// TIA Portal V18 export
FUNCTION "TEMPLATE--v1.1--05_Output Feedback" : Void   // FC6, F_FBD
TITLE = Manage Safety Outputs
{ S7_Optimized_Access := 'TRUE' }
// v1.0 First Emission
// v1.1 Added 03_FDBACK_RAW reference
   VAR_TEMP
      DU_EX : Bool;
      ISPC_EX : Bool;
      ZONE_EX : Bool;
   END_VAR
BEGIN

REGION Network 1: !!NetworkComment$$ 1c -1i -1q
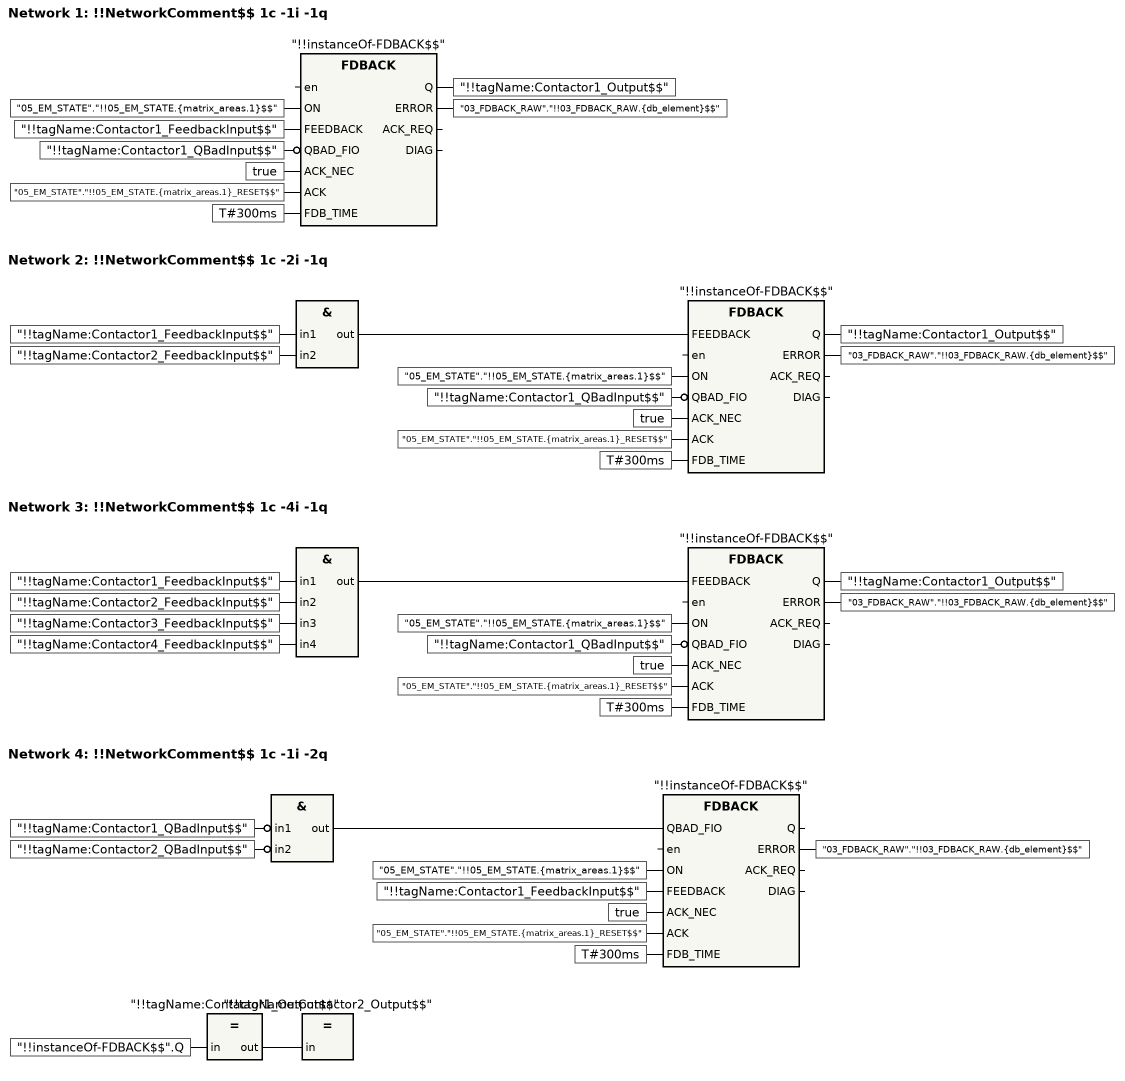
   "!!instanceOf-FDBACK$$"(ON := "05_EM_STATE"."!!05_EM_STATE.{matrix_areas.1}$$",   // FDBACK
                           FEEDBACK := "!!tagName:Contactor1_FeedbackInput$$",
                           QBAD_FIO := NOT "!!tagName:Contactor1_QBadInput$$",
                           ACK_NEC := true,
                           ACK := "05_EM_STATE"."!!05_EM_STATE.{matrix_areas.1}_RESET$$",
                           FDB_TIME := T#300ms,
                           Q => "!!tagName:Contactor1_Output$$",
                           ERROR => "03_FDBACK_RAW"."!!03_FDBACK_RAW.{db_element}$$");
END_REGION

REGION Network 2: !!NetworkComment$$ 1c -2i -1q
   "!!instanceOf-FDBACK$$"(FEEDBACK := "!!tagName:Contactor1_FeedbackInput$$" AND "!!tagName:Contactor2_FeedbackInput$$",   // FDBACK
                           ON := "05_EM_STATE"."!!05_EM_STATE.{matrix_areas.1}$$",
                           QBAD_FIO := NOT "!!tagName:Contactor1_QBadInput$$",
                           ACK_NEC := true,
                           ACK := "05_EM_STATE"."!!05_EM_STATE.{matrix_areas.1}_RESET$$",
                           FDB_TIME := T#300ms,
                           Q => "!!tagName:Contactor1_Output$$",
                           ERROR => "03_FDBACK_RAW"."!!03_FDBACK_RAW.{db_element}$$");
END_REGION

REGION Network 3: !!NetworkComment$$ 1c -4i -1q
   "!!instanceOf-FDBACK$$"(FEEDBACK := "!!tagName:Contactor1_FeedbackInput$$" AND "!!tagName:Contactor2_FeedbackInput$$" AND "!!tagName:Contactor3_FeedbackInput$$" AND "!!tagName:Contactor4_FeedbackInput$$",   // FDBACK
                           ON := "05_EM_STATE"."!!05_EM_STATE.{matrix_areas.1}$$",
                           QBAD_FIO := NOT "!!tagName:Contactor1_QBadInput$$",
                           ACK_NEC := true,
                           ACK := "05_EM_STATE"."!!05_EM_STATE.{matrix_areas.1}_RESET$$",
                           FDB_TIME := T#300ms,
                           Q => "!!tagName:Contactor1_Output$$",
                           ERROR => "03_FDBACK_RAW"."!!03_FDBACK_RAW.{db_element}$$");
END_REGION

REGION Network 4: !!NetworkComment$$ 1c -1i -2q
   "!!instanceOf-FDBACK$$"(QBAD_FIO := NOT "!!tagName:Contactor1_QBadInput$$" AND NOT "!!tagName:Contactor2_QBadInput$$",   // FDBACK
                           ON := "05_EM_STATE"."!!05_EM_STATE.{matrix_areas.1}$$",
                           FEEDBACK := "!!tagName:Contactor1_FeedbackInput$$",
                           ACK_NEC := true,
                           ACK := "05_EM_STATE"."!!05_EM_STATE.{matrix_areas.1}_RESET$$",
                           FDB_TIME := T#300ms,
                           ERROR => "03_FDBACK_RAW"."!!03_FDBACK_RAW.{db_element}$$");
   "!!tagName:Contactor1_Output$$" := "!!instanceOf-FDBACK$$".Q;
   "!!tagName:Contactor2_Output$$" := "!!instanceOf-FDBACK$$".Q;
END_REGION

REGION Network 5: !!NetworkComment$$ 1c -2i -2q
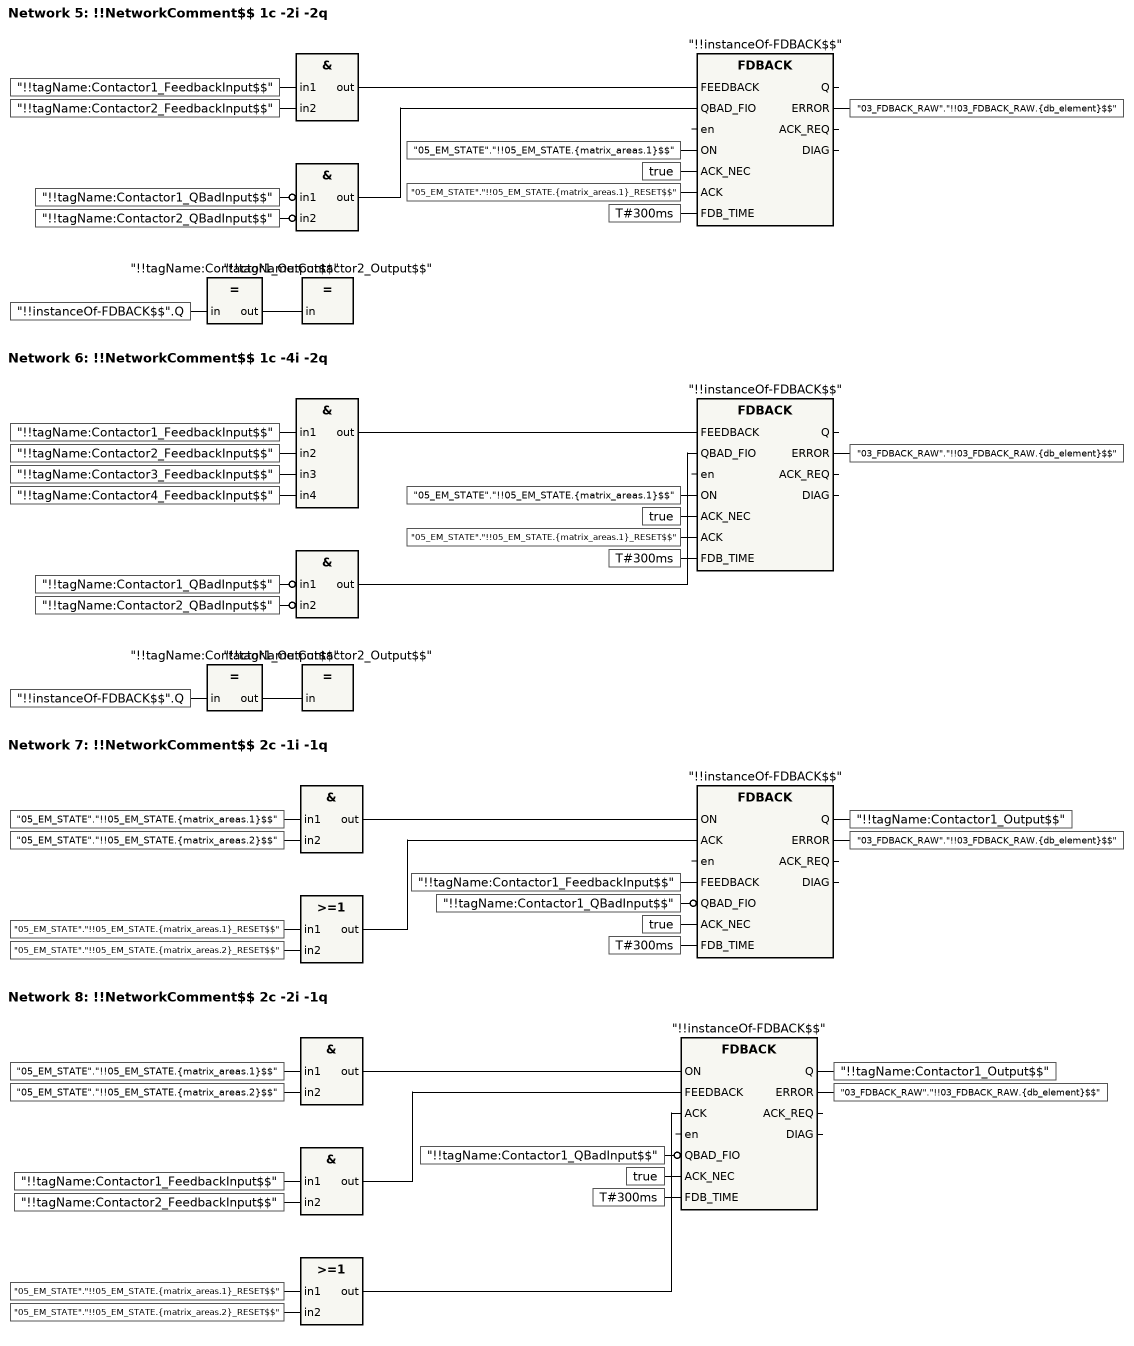
   "!!instanceOf-FDBACK$$"(FEEDBACK := "!!tagName:Contactor1_FeedbackInput$$" AND "!!tagName:Contactor2_FeedbackInput$$",   // FDBACK
                           QBAD_FIO := NOT "!!tagName:Contactor1_QBadInput$$" AND NOT "!!tagName:Contactor2_QBadInput$$",
                           ON := "05_EM_STATE"."!!05_EM_STATE.{matrix_areas.1}$$",
                           ACK_NEC := true,
                           ACK := "05_EM_STATE"."!!05_EM_STATE.{matrix_areas.1}_RESET$$",
                           FDB_TIME := T#300ms,
                           ERROR => "03_FDBACK_RAW"."!!03_FDBACK_RAW.{db_element}$$");
   "!!tagName:Contactor1_Output$$" := "!!instanceOf-FDBACK$$".Q;
   "!!tagName:Contactor2_Output$$" := "!!instanceOf-FDBACK$$".Q;
END_REGION

REGION Network 6: !!NetworkComment$$ 1c -4i -2q
   "!!instanceOf-FDBACK$$"(FEEDBACK := "!!tagName:Contactor1_FeedbackInput$$" AND "!!tagName:Contactor2_FeedbackInput$$" AND "!!tagName:Contactor3_FeedbackInput$$" AND "!!tagName:Contactor4_FeedbackInput$$",   // FDBACK
                           QBAD_FIO := NOT "!!tagName:Contactor1_QBadInput$$" AND NOT "!!tagName:Contactor2_QBadInput$$",
                           ON := "05_EM_STATE"."!!05_EM_STATE.{matrix_areas.1}$$",
                           ACK_NEC := true,
                           ACK := "05_EM_STATE"."!!05_EM_STATE.{matrix_areas.1}_RESET$$",
                           FDB_TIME := T#300ms,
                           ERROR => "03_FDBACK_RAW"."!!03_FDBACK_RAW.{db_element}$$");
   "!!tagName:Contactor1_Output$$" := "!!instanceOf-FDBACK$$".Q;
   "!!tagName:Contactor2_Output$$" := "!!instanceOf-FDBACK$$".Q;
END_REGION

REGION Network 7: !!NetworkComment$$ 2c -1i -1q
   "!!instanceOf-FDBACK$$"(ON := "05_EM_STATE"."!!05_EM_STATE.{matrix_areas.1}$$" AND "05_EM_STATE"."!!05_EM_STATE.{matrix_areas.2}$$",   // FDBACK
                           ACK := "05_EM_STATE"."!!05_EM_STATE.{matrix_areas.1}_RESET$$" OR "05_EM_STATE"."!!05_EM_STATE.{matrix_areas.2}_RESET$$",
                           FEEDBACK := "!!tagName:Contactor1_FeedbackInput$$",
                           QBAD_FIO := NOT "!!tagName:Contactor1_QBadInput$$",
                           ACK_NEC := true,
                           FDB_TIME := T#300ms,
                           Q => "!!tagName:Contactor1_Output$$",
                           ERROR => "03_FDBACK_RAW"."!!03_FDBACK_RAW.{db_element}$$");
END_REGION

REGION Network 8: !!NetworkComment$$ 2c -2i -1q
   "!!instanceOf-FDBACK$$"(ON := "05_EM_STATE"."!!05_EM_STATE.{matrix_areas.1}$$" AND "05_EM_STATE"."!!05_EM_STATE.{matrix_areas.2}$$",   // FDBACK
                           FEEDBACK := "!!tagName:Contactor1_FeedbackInput$$" AND "!!tagName:Contactor2_FeedbackInput$$",
                           ACK := "05_EM_STATE"."!!05_EM_STATE.{matrix_areas.1}_RESET$$" OR "05_EM_STATE"."!!05_EM_STATE.{matrix_areas.2}_RESET$$",
                           QBAD_FIO := NOT "!!tagName:Contactor1_QBadInput$$",
                           ACK_NEC := true,
                           FDB_TIME := T#300ms,
                           Q => "!!tagName:Contactor1_Output$$",
                           ERROR => "03_FDBACK_RAW"."!!03_FDBACK_RAW.{db_element}$$");
END_REGION

REGION Network 9: !!NetworkComment$$ 1c -4i -1q
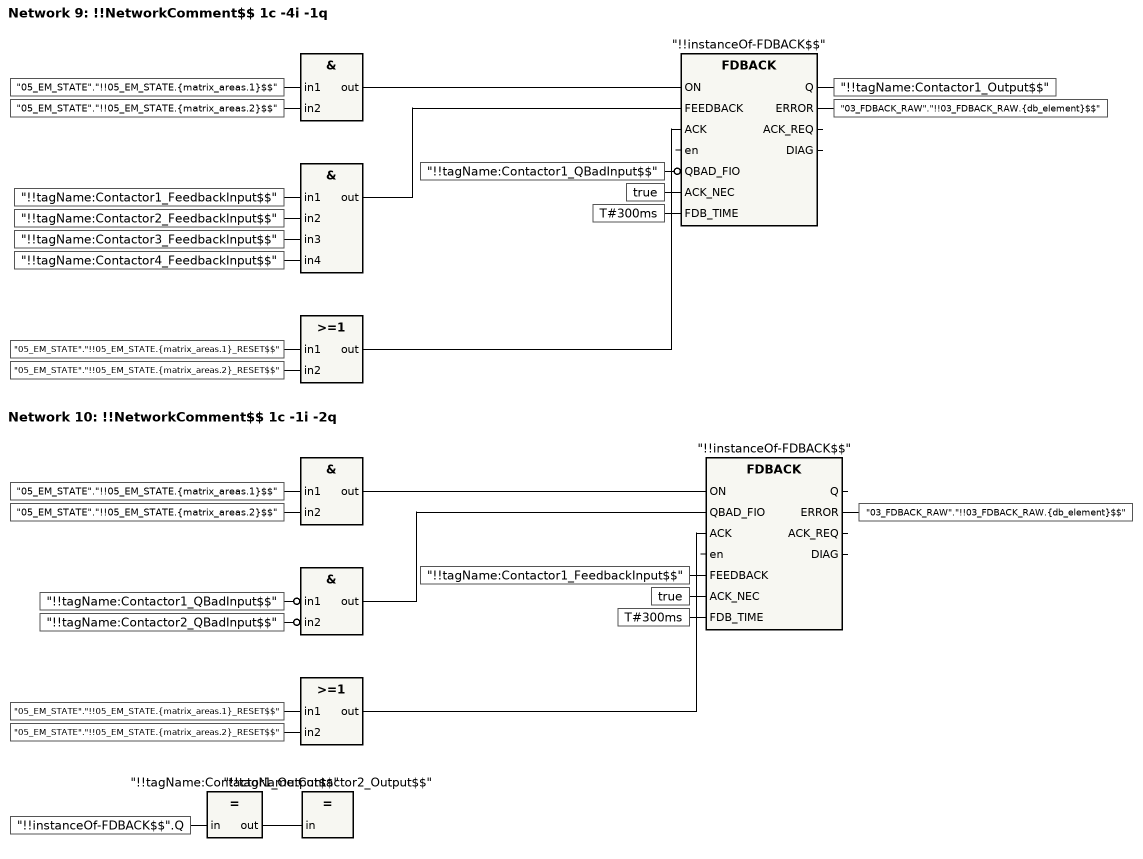
   "!!instanceOf-FDBACK$$"(ON := "05_EM_STATE"."!!05_EM_STATE.{matrix_areas.1}$$" AND "05_EM_STATE"."!!05_EM_STATE.{matrix_areas.2}$$",   // FDBACK
                           FEEDBACK := "!!tagName:Contactor1_FeedbackInput$$" AND "!!tagName:Contactor2_FeedbackInput$$" AND "!!tagName:Contactor3_FeedbackInput$$" AND "!!tagName:Contactor4_FeedbackInput$$",
                           ACK := "05_EM_STATE"."!!05_EM_STATE.{matrix_areas.1}_RESET$$" OR "05_EM_STATE"."!!05_EM_STATE.{matrix_areas.2}_RESET$$",
                           QBAD_FIO := NOT "!!tagName:Contactor1_QBadInput$$",
                           ACK_NEC := true,
                           FDB_TIME := T#300ms,
                           Q => "!!tagName:Contactor1_Output$$",
                           ERROR => "03_FDBACK_RAW"."!!03_FDBACK_RAW.{db_element}$$");
END_REGION

REGION Network 10: !!NetworkComment$$ 1c -1i -2q
   "!!instanceOf-FDBACK$$"(ON := "05_EM_STATE"."!!05_EM_STATE.{matrix_areas.1}$$" AND "05_EM_STATE"."!!05_EM_STATE.{matrix_areas.2}$$",   // FDBACK
                           QBAD_FIO := NOT "!!tagName:Contactor1_QBadInput$$" AND NOT "!!tagName:Contactor2_QBadInput$$",
                           ACK := "05_EM_STATE"."!!05_EM_STATE.{matrix_areas.1}_RESET$$" OR "05_EM_STATE"."!!05_EM_STATE.{matrix_areas.2}_RESET$$",
                           FEEDBACK := "!!tagName:Contactor1_FeedbackInput$$",
                           ACK_NEC := true,
                           FDB_TIME := T#300ms,
                           ERROR => "03_FDBACK_RAW"."!!03_FDBACK_RAW.{db_element}$$");
   "!!tagName:Contactor1_Output$$" := "!!instanceOf-FDBACK$$".Q;
   "!!tagName:Contactor2_Output$$" := "!!instanceOf-FDBACK$$".Q;
END_REGION

REGION Network 11: !!NetworkComment$$ 1c -2i -2q
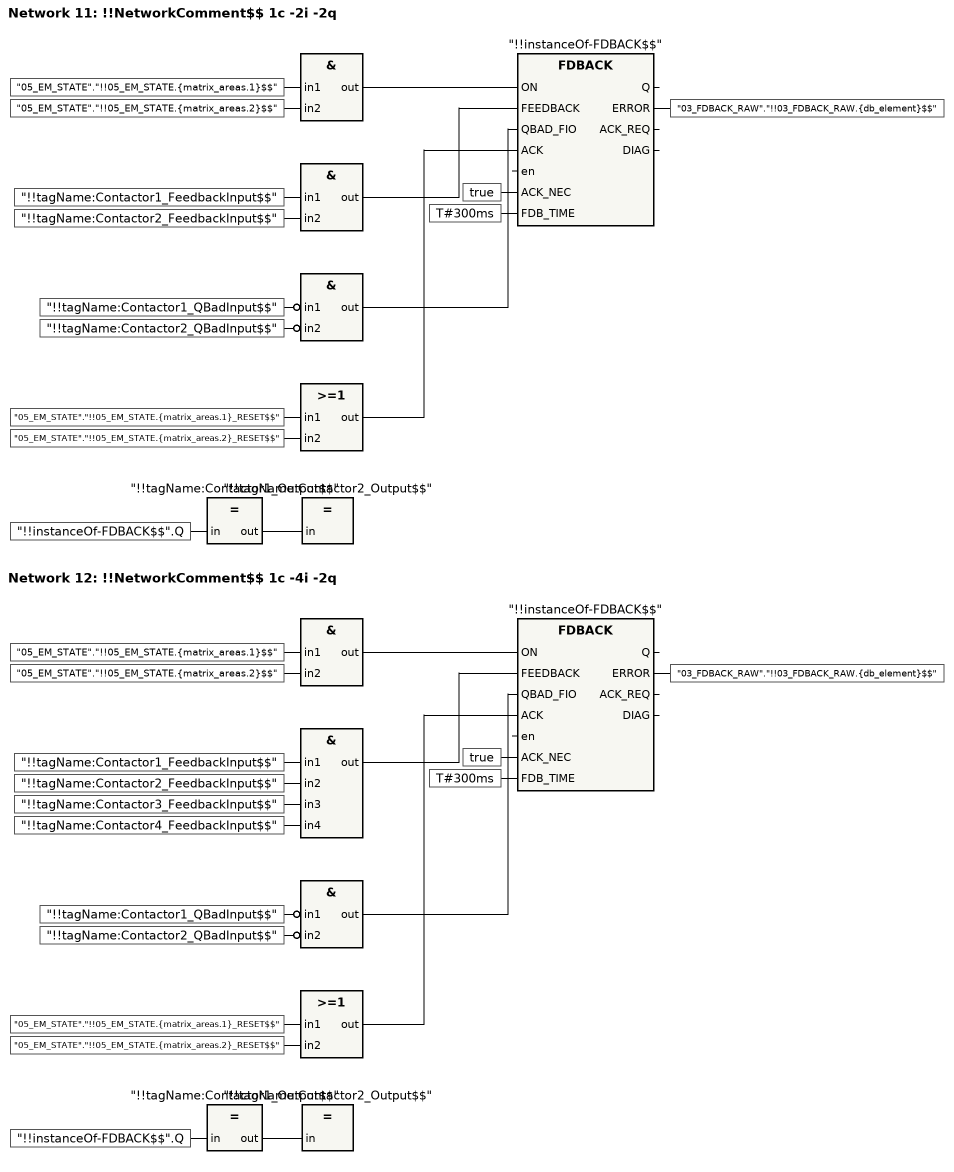
   "!!instanceOf-FDBACK$$"(ON := "05_EM_STATE"."!!05_EM_STATE.{matrix_areas.1}$$" AND "05_EM_STATE"."!!05_EM_STATE.{matrix_areas.2}$$",   // FDBACK
                           FEEDBACK := "!!tagName:Contactor1_FeedbackInput$$" AND "!!tagName:Contactor2_FeedbackInput$$",
                           QBAD_FIO := NOT "!!tagName:Contactor1_QBadInput$$" AND NOT "!!tagName:Contactor2_QBadInput$$",
                           ACK := "05_EM_STATE"."!!05_EM_STATE.{matrix_areas.1}_RESET$$" OR "05_EM_STATE"."!!05_EM_STATE.{matrix_areas.2}_RESET$$",
                           ACK_NEC := true,
                           FDB_TIME := T#300ms,
                           ERROR => "03_FDBACK_RAW"."!!03_FDBACK_RAW.{db_element}$$");
   "!!tagName:Contactor1_Output$$" := "!!instanceOf-FDBACK$$".Q;
   "!!tagName:Contactor2_Output$$" := "!!instanceOf-FDBACK$$".Q;
END_REGION

REGION Network 12: !!NetworkComment$$ 1c -4i -2q
   "!!instanceOf-FDBACK$$"(ON := "05_EM_STATE"."!!05_EM_STATE.{matrix_areas.1}$$" AND "05_EM_STATE"."!!05_EM_STATE.{matrix_areas.2}$$",   // FDBACK
                           FEEDBACK := "!!tagName:Contactor1_FeedbackInput$$" AND "!!tagName:Contactor2_FeedbackInput$$" AND "!!tagName:Contactor3_FeedbackInput$$" AND "!!tagName:Contactor4_FeedbackInput$$",
                           QBAD_FIO := NOT "!!tagName:Contactor1_QBadInput$$" AND NOT "!!tagName:Contactor2_QBadInput$$",
                           ACK := "05_EM_STATE"."!!05_EM_STATE.{matrix_areas.1}_RESET$$" OR "05_EM_STATE"."!!05_EM_STATE.{matrix_areas.2}_RESET$$",
                           ACK_NEC := true,
                           FDB_TIME := T#300ms,
                           ERROR => "03_FDBACK_RAW"."!!03_FDBACK_RAW.{db_element}$$");
   "!!tagName:Contactor1_Output$$" := "!!instanceOf-FDBACK$$".Q;
   "!!tagName:Contactor2_Output$$" := "!!instanceOf-FDBACK$$".Q;
END_REGION
END_FUNCTION
